Fanuc KAREL source: kb00181.KL

-- PROVISIONAL review KL for V1013-1; original PC SHA256 8de52542c61516fcf50995f98b897823ad7a41341325c4fd7a7137bdec20b705
-- Incomplete behavior may be omitted. Consult companion uncertainty JSON. Do not deploy.
PROGRAM KB00181
%NOLOCKGROUP
BEGIN
  -- UNRESOLVED_PC offsets 5-12; opcodes 9D,23
  -- UNRESOLVED_PC offsets 17-27; opcodes 27,22,31
  -- UNRESOLVED_PC offsets 32-36; opcodes 7F
END KB00181
